// TIA Portal V20 export
DATA_BLOCK "BK01"   // DB222
// stored: MemoryReserve 100
   VAR
      "X10-1 LEFT UNWINDER EXPEL BACKWARD" : Bool;
      "X11-1 RIGHT UNWINDER EXPEL BACKWARD" : Bool;
      "X12-1 UW SUPPORT UNIT TRANSFER BACKWARD" : Bool;
      "X13-1 ELECTRODE SHAFT SUPPORTER DOWN" : Bool;
      "X14-1 LEFT TENSION CHECK SENSOR" : Bool;
      "X15-1 ELECTRODE FIX LEFT TOP PRESSURE SWITCH" : Bool;
      "X16-1 SPARE" : Bool;
      "X17-1 SPARE" : Bool;
      "X10-2 LEFT UNWINDER EXPEL FORWARD" : Bool;
      "X11-2 RIGHT UNWINDER EXPEL FORWARD" : Bool;
      "X12-2 UW SUPPORT UNIT TRANSFER FORWARD" : Bool;
      "X13-2 ELECTRODE SHAFT SUPPORTER UP" : Bool;
      "X14-2 RIGHT TENSION CHECK SENSOR" : Bool;
      "X15-2 ELECTRODE FIX LEFT BTM PRESSURE SWITCH" : Bool;
      "X16-2 SPARE" : Bool;
      "X17-2 SPARE" : Bool;
   END_VAR
BEGIN
END_DATA_BLOCK
